// TIA Portal V17 export
// export: Created 2025-03-07T09:18:48.0864435Z, ExportSetting WithDefaults, DisplayName Totally Integrated Automation Portal, DisplayVersion V17 Update 8, DisplayName TIA Portal Openness, DisplayVersion V17 Update 8, DisplayName TIA Portal Version Control Interface, DisplayVersion V17, DisplayName SINAMICS Startdrive Advanced, DisplayVersion V17 SP2, DisplayName SINAMICS Startdrive G110M, G120, G120C, G120D, G120P, G115D, DisplayVersion V17 SP2, DisplayName SINAMICS Startdrive G130, G150, S120, S150, SINAMICS MV, S210, DisplayVersion V17 SP2, DisplayName STEP 7 Professional, DisplayVersion V17 Update 8, DisplayName SINUMERIK ONE STEP 7 Toolbox, DisplayVersion V17 Update 12, DisplayName SINUMERIK 840D sl STEP 7 Toolbox, DisplayVersion V17 Update 12, DisplayName STEP 7 Safety, DisplayVersion V17 Update 6, DisplayName WinCC Advanced, DisplayVersion V17 Update 8
FUNCTION_BLOCK "FB6500_CYLINDER"   // FB6500, LAD
{ S7_Optimized_Access := 'FALSE' }
AUTHOR : ETXETAR
VERSION : 1.0
// stored: AutoNumber false, IsIECCheckEnabled false, SetENOAutomatically false, UDAEnableTagReadback false
   VAR_INPUT
      OPTIONS_0 : Byte := 2#0000_0000;   // OPTIONS 0
      ADVANCED_1_I : Bool;   // ADVANCED 1 INPUT
      ADVANCED_2_I : Bool;   // ADVANCED 2 INPUT
      ADVANCED_3_I : Bool;   // ADVANCED 3 INPUT
      ADVANCED_4_I : Bool;   // ADVANCED 4 INPUT
      RETURNED_1_I : Bool;   // OPEN 1 INPUT
      RETURNED_2_I : Bool;   // OPEN 2 INPUT
      RETURNED_3_I : Bool;   // OPEN 3 INPUT
      RETURNED_4_I : Bool;   // OPEN 4 INPUT
      ADVANCE_CONDITIONS : Bool;   // ADVANCE CONDITIONS
      RETURN_CONDITIONS : Bool;   // OPEN CONDITIONS
      HMI_LINE_REQUEST : Bool;   // HMI LINE REQUEST
      ADVANCE_AUTO_REQUEST : Bool;   // AUTO ADVANCE REQUEST
      RETURN_AUTO_REQUEST : Bool;   // AUTO OPEN REQUEST
      UNIT_ALARM : UInt;   // UNIT NUMBER MIN. NUMBER=1 MAX. NUMBER=4
      STATION_ALARM : UInt;   // STATION NUMBER MIN. NUMBER=0 MAX. NUMBER=4
   END_VAR
   VAR_OUTPUT
      ADVANCED : Bool;   // ADVANCED
      RETURNED : Bool;   // OPEN STATUS
      ADVANCED_1_ALARM : Bool;   // ADVANCED 1 ALARM
      ADVANCED_2_ALARM : Bool;   // ADVANCED 2 ALARM
      ADVANCED_3_ALARM : Bool;   // ADVANCED 3 ALARM
      ADVANCED_4_ALARM : Bool;   // ADVANCED 4 ALARM
      RETURNED_1_ALARM : Bool;   // OPEN 1 ALARM
      RETURNED_2_ALARM : Bool;   // OPEN 2 ALARM
      RETURNED_3_ALARM : Bool;   // OPEN 3 ALARM
      RETURNED_4_ALARM : Bool;   // OPEN 4 ALARM
      HMI_MOTION_EXECUTABILITY_LEFT : Bool;   // HMI MOTION EXECUTABILITY LEFT
      HMI_MOTION_EXECUTABILITY_RIGHT : Bool;   // HMI MOTION EXECUTABILITY RIGHT
      HMI_MOTION_END_POS_LEFT : Bool;   // HMI MOTION END POSITION LEFT
      HMI_MOTION_END_POS_RIGHT : Bool;   // HMI MOTION END POSITION RIGHT
      HMI_MOTION_ACTIVE_LEFT : Bool;   // HMI MOTION ACTIVE LEFT
      HMI_MOTION_ACTIVE_RIGHT : Bool;   // HMI MOTION ACTIVE RIGHT
      ADVANCE : Bool;   // ADVANCE OUTPUT
      "RETURN" : Bool;   // OPEN OUTPUT
   END_VAR
   VAR DB_SPECIFIC
      CYL { S7_SetPoint := 'True'} : "ADVANCE_RETURN_CYL_CLADDING";
      TIMER_ADVANCED { S7_SetPoint := 'True'} : TON_TIME;   // ADVANCED TIMER
      TIMER_RETURNED { S7_SetPoint := 'True'} : TON_TIME;   // OPENED TIMER
      TIMER_SIMULTANEITY { S7_SetPoint := 'True'} : TON_TIME;   // SIMULTANEITY TIMER
      TIMER_TIME_EXCEEDED { S7_SetPoint := 'True'} : TON_TIME;   // TIME EXCEEDED TIMER
   END_VAR
   VAR_TEMP
      INPUTS_MASK : Byte;   // INPUTS_MASK
      O_BYTE_0 : Struct   // OPTIONS BYTE 0
         ADVANCED_INPUT_1 : Bool;   // ADVANCED INPUT 1 OPTION
         ADVANCED_INPUT_2 : Bool;   // ADVANCED INPUT 2 OPTION
         ADVANCED_INPUT_3 : Bool;   // ADVANCED INPUT 3 OPTION
         ADVANCED_INPUT_4 : Bool;   // ADVANCED INPUT 4 OPTION
         RETURNED_INPUT_1 : Bool;   // OPEN INPUT 1 OPTION
         RETURNED_INPUT_2 : Bool;   // OPEN INPUT 2 OPTION
         RETURNED_INPUT_3 : Bool;   // OPEN INPUT 3 OPTION
         RETURNED_INPUT_4 : Bool;   // OPEN INPUT 4 OPTION
      END_STRUCT;
      DB_NUMBER : DInt;   // DB NUMBER FOR ALARM AND HELP DECODING
   END_VAR
   // TIMER_ADVANCED.PT := T#100MS;
   // TIMER_RETURNED.PT := T#300MS;
   // TIMER_SIMULTANEITY.PT := T#100MS;
   // TIMER_TIME_EXCEEDED.PT := T#8S;
   VAR_TEMP   // added for the SCL form of the ladder/FBD networks
      _w1 : Bool;
      _w2 : Bool;
   END_VAR
BEGIN

NETWORK
TITLE = READ INSTANCE DB
      L     DINO;
      +     10#800000;
      T     #DB_NUMBER;


REGION Network 2: OPTIONS
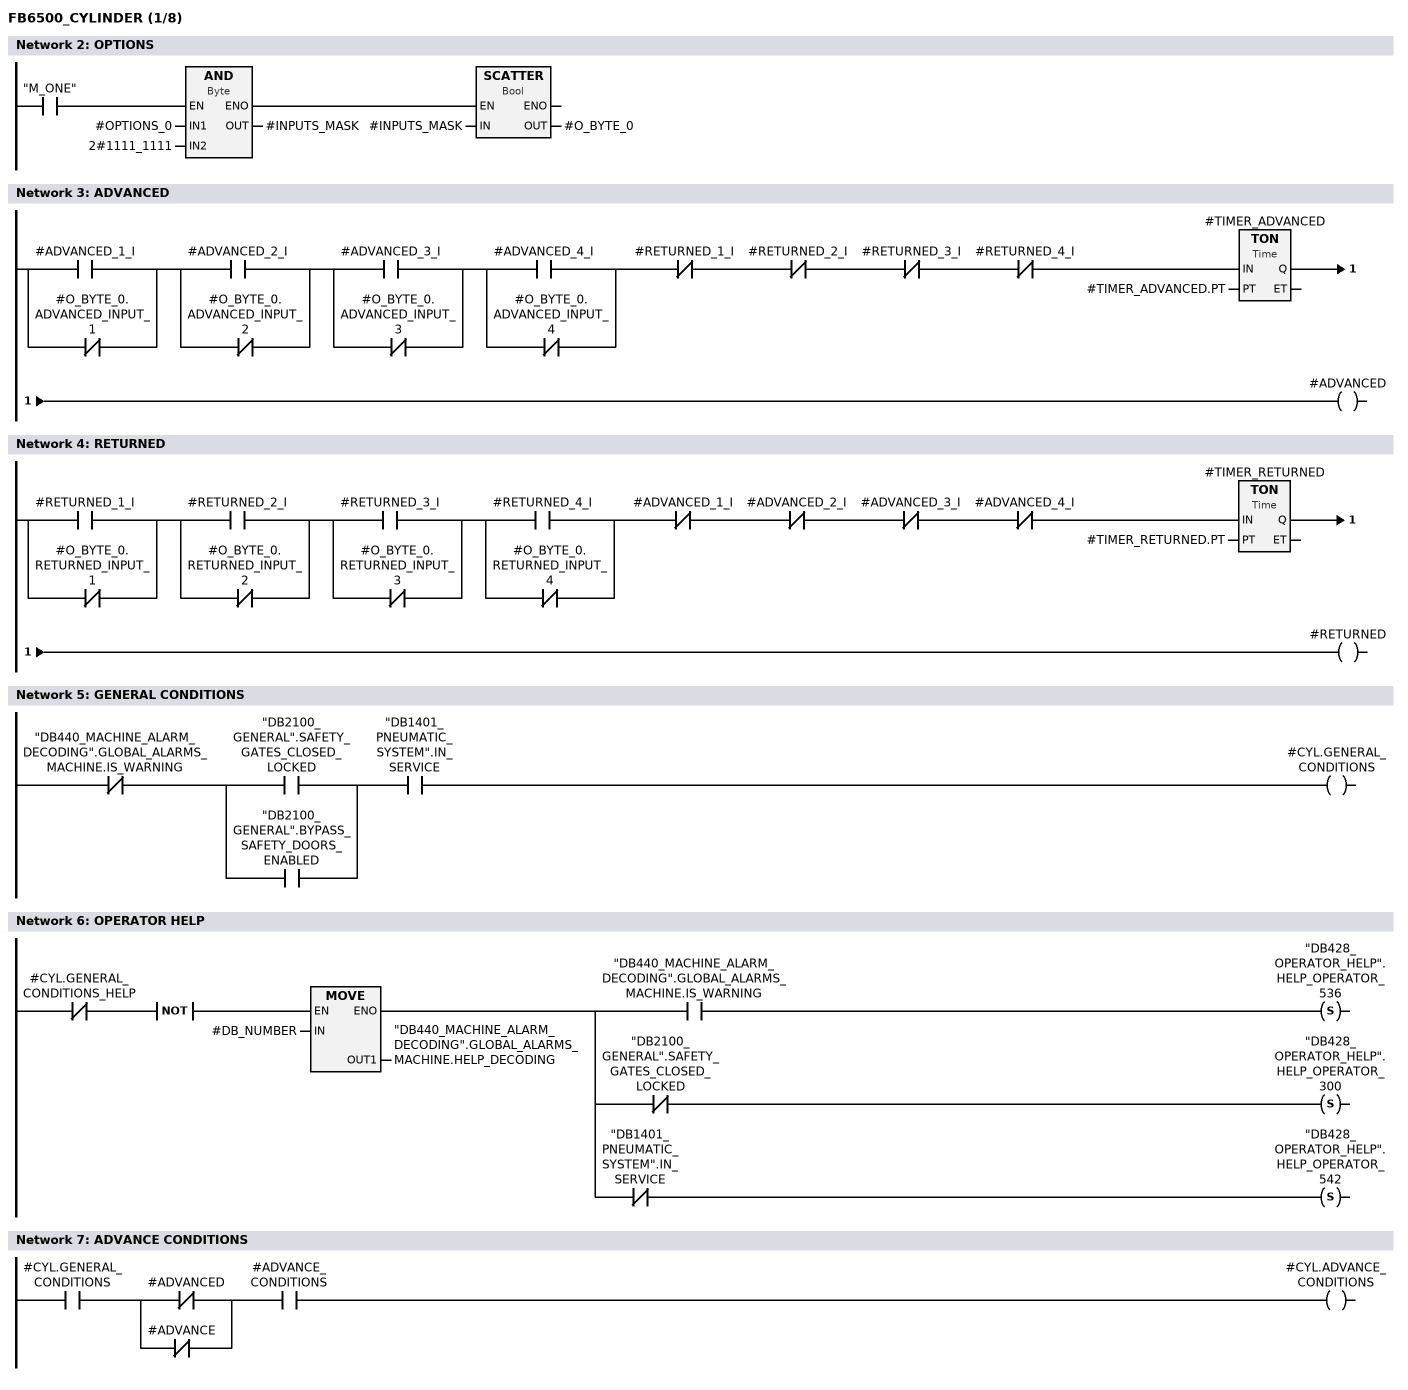
   RUNG wire#powerrail
      Contact( "M_ONE" )
      { S7_Templates := "SrcType := Byte"; S7_GenerateENO := "TRUE" } And(in1 := #OPTIONS_0, in2 := 2#1111_1111, out => #INPUTS_MASK)
      { S7_Templates := "[dest_type := Bool, src_type := Byte]" } SCATTER(IN := #INPUTS_MASK, OUT => #O_BYTE_0)
   END_RUNG
   // the same network as SCL:
   IF "M_ONE" THEN
       #INPUTS_MASK := #OPTIONS_0 AND 2#1111_1111;
       SCATTER(IN := #INPUTS_MASK, OUT => #O_BYTE_0);
   END_IF;
END_REGION

REGION Network 3: ADVANCED
   RUNG wire#powerrail
      Contact( #ADVANCED_1_I )
      wire#w1
      Contact( #ADVANCED_2_I )
      wire#w2
      Contact( #ADVANCED_3_I )
      wire#w3
      Contact( #ADVANCED_4_I )
      wire#w4
      I_Contact( #RETURNED_1_I )
      I_Contact( #RETURNED_2_I )
      I_Contact( #RETURNED_3_I )
      I_Contact( #RETURNED_4_I )
      { S7_Templates := "time_type := Time" } #TIMER_ADVANCED.TON(pt := #TIMER_ADVANCED.PT, et =>)
      Coil( #ADVANCED )
   END_RUNG
   RUNG wire#powerrail
      I_Contact( #O_BYTE_0.ADVANCED_INPUT_1 )
   END_RUNG wire#w1
   RUNG wire#w1
      I_Contact( #O_BYTE_0.ADVANCED_INPUT_2 )
   END_RUNG wire#w2
   RUNG wire#w2
      I_Contact( #O_BYTE_0.ADVANCED_INPUT_3 )
   END_RUNG wire#w3
   RUNG wire#w3
      I_Contact( #O_BYTE_0.ADVANCED_INPUT_4 )
   END_RUNG wire#w4
   // the same network as SCL:
   #TIMER_ADVANCED(IN := (#ADVANCED_1_I OR NOT #O_BYTE_0.ADVANCED_INPUT_1) AND (#ADVANCED_2_I OR NOT #O_BYTE_0.ADVANCED_INPUT_2) AND (#ADVANCED_3_I OR NOT #O_BYTE_0.ADVANCED_INPUT_3) AND (#ADVANCED_4_I OR NOT #O_BYTE_0.ADVANCED_INPUT_4) AND NOT #RETURNED_1_I AND NOT #RETURNED_2_I AND NOT #RETURNED_3_I AND NOT #RETURNED_4_I,   // TON
                   PT := #TIMER_ADVANCED.PT);
   #ADVANCED := #TIMER_ADVANCED.Q;
END_REGION

REGION Network 4: RETURNED
   RUNG wire#powerrail
      Contact( #RETURNED_1_I )
      wire#w1
      Contact( #RETURNED_2_I )
      wire#w2
      Contact( #RETURNED_3_I )
      wire#w3
      Contact( #RETURNED_4_I )
      wire#w4
      I_Contact( #ADVANCED_1_I )
      I_Contact( #ADVANCED_2_I )
      I_Contact( #ADVANCED_3_I )
      I_Contact( #ADVANCED_4_I )
      { S7_Templates := "time_type := Time" } #TIMER_RETURNED.TON(pt := #TIMER_RETURNED.PT, et =>)
      Coil( #RETURNED )
   END_RUNG
   RUNG wire#powerrail
      I_Contact( #O_BYTE_0.RETURNED_INPUT_1 )
   END_RUNG wire#w1
   RUNG wire#w1
      I_Contact( #O_BYTE_0.RETURNED_INPUT_2 )
   END_RUNG wire#w2
   RUNG wire#w2
      I_Contact( #O_BYTE_0.RETURNED_INPUT_3 )
   END_RUNG wire#w3
   RUNG wire#w3
      I_Contact( #O_BYTE_0.RETURNED_INPUT_4 )
   END_RUNG wire#w4
   // the same network as SCL:
   #TIMER_RETURNED(IN := (#RETURNED_1_I OR NOT #O_BYTE_0.RETURNED_INPUT_1) AND (#RETURNED_2_I OR NOT #O_BYTE_0.RETURNED_INPUT_2) AND (#RETURNED_3_I OR NOT #O_BYTE_0.RETURNED_INPUT_3) AND (#RETURNED_4_I OR NOT #O_BYTE_0.RETURNED_INPUT_4) AND NOT #ADVANCED_1_I AND NOT #ADVANCED_2_I AND NOT #ADVANCED_3_I AND NOT #ADVANCED_4_I,   // TON
                   PT := #TIMER_RETURNED.PT);
   #RETURNED := #TIMER_RETURNED.Q;
END_REGION

REGION Network 5: GENERAL CONDITIONS
   RUNG wire#powerrail
      I_Contact( "DB440_MACHINE_ALARM_DECODING".GLOBAL_ALARMS_MACHINE.IS_WARNING )
      wire#w1
      Contact( "DB2100_GENERAL".SAFETY_GATES_CLOSED_LOCKED )
      wire#w2
      Contact( "DB1401_PNEUMATIC_SYSTEM".IN_SERVICE )
      Coil( #CYL.GENERAL_CONDITIONS )
   END_RUNG
   RUNG wire#w1
      Contact( "DB2100_GENERAL".BYPASS_SAFETY_DOORS_ENABLED )
   END_RUNG wire#w2
   // the same network as SCL:
   #CYL.GENERAL_CONDITIONS := NOT "DB440_MACHINE_ALARM_DECODING".GLOBAL_ALARMS_MACHINE.IS_WARNING AND ("DB2100_GENERAL".SAFETY_GATES_CLOSED_LOCKED OR "DB2100_GENERAL".BYPASS_SAFETY_DOORS_ENABLED) AND "DB1401_PNEUMATIC_SYSTEM".IN_SERVICE;
END_REGION

REGION Network 6: OPERATOR HELP
   RUNG wire#powerrail
      I_Contact( #CYL.GENERAL_CONDITIONS_HELP )
      Not()
      { S7_GenerateENO := "TRUE" } Move(in := #DB_NUMBER, out1 => "DB440_MACHINE_ALARM_DECODING".GLOBAL_ALARMS_MACHINE.HELP_DECODING)
      wire#w1
      Contact( "DB440_MACHINE_ALARM_DECODING".GLOBAL_ALARMS_MACHINE.IS_WARNING )
      S_Coil( "DB428_OPERATOR_HELP".HELP_OPERATOR_536 )
   END_RUNG
   RUNG wire#w1
      I_Contact( "DB2100_GENERAL".SAFETY_GATES_CLOSED_LOCKED )
      S_Coil( "DB428_OPERATOR_HELP".HELP_OPERATOR_300 )
   END_RUNG
   RUNG wire#w1
      I_Contact( "DB1401_PNEUMATIC_SYSTEM".IN_SERVICE )
      S_Coil( "DB428_OPERATOR_HELP".HELP_OPERATOR_542 )
   END_RUNG
   // the same network as SCL:
   // ENO of a box is taken as its EN; it also drops when the box reports an error
   #_w1 := NOT (NOT #CYL.GENERAL_CONDITIONS_HELP);
   IF #_w1 THEN "DB440_MACHINE_ALARM_DECODING".GLOBAL_ALARMS_MACHINE.HELP_DECODING := #DB_NUMBER; END_IF;
   IF #_w1 AND "DB440_MACHINE_ALARM_DECODING".GLOBAL_ALARMS_MACHINE.IS_WARNING THEN
       "DB428_OPERATOR_HELP".HELP_OPERATOR_536 := TRUE;
   END_IF;
   IF #_w1 AND NOT "DB2100_GENERAL".SAFETY_GATES_CLOSED_LOCKED THEN
       "DB428_OPERATOR_HELP".HELP_OPERATOR_300 := TRUE;
   END_IF;
   IF #_w1 AND NOT "DB1401_PNEUMATIC_SYSTEM".IN_SERVICE THEN
       "DB428_OPERATOR_HELP".HELP_OPERATOR_542 := TRUE;
   END_IF;
END_REGION

REGION Network 7: ADVANCE CONDITIONS
   RUNG wire#powerrail
      Contact( #CYL.GENERAL_CONDITIONS )
      wire#w1
      I_Contact( #ADVANCED )
      wire#w2
      Contact( #ADVANCE_CONDITIONS )
      Coil( #CYL.ADVANCE_CONDITIONS )
   END_RUNG
   RUNG wire#w1
      I_Contact( #ADVANCE )
   END_RUNG wire#w2
   // the same network as SCL:
   #CYL.ADVANCE_CONDITIONS := #CYL.GENERAL_CONDITIONS AND (NOT #ADVANCED OR NOT #ADVANCE) AND #ADVANCE_CONDITIONS;
END_REGION

REGION Network 8: OPERATOR HELP
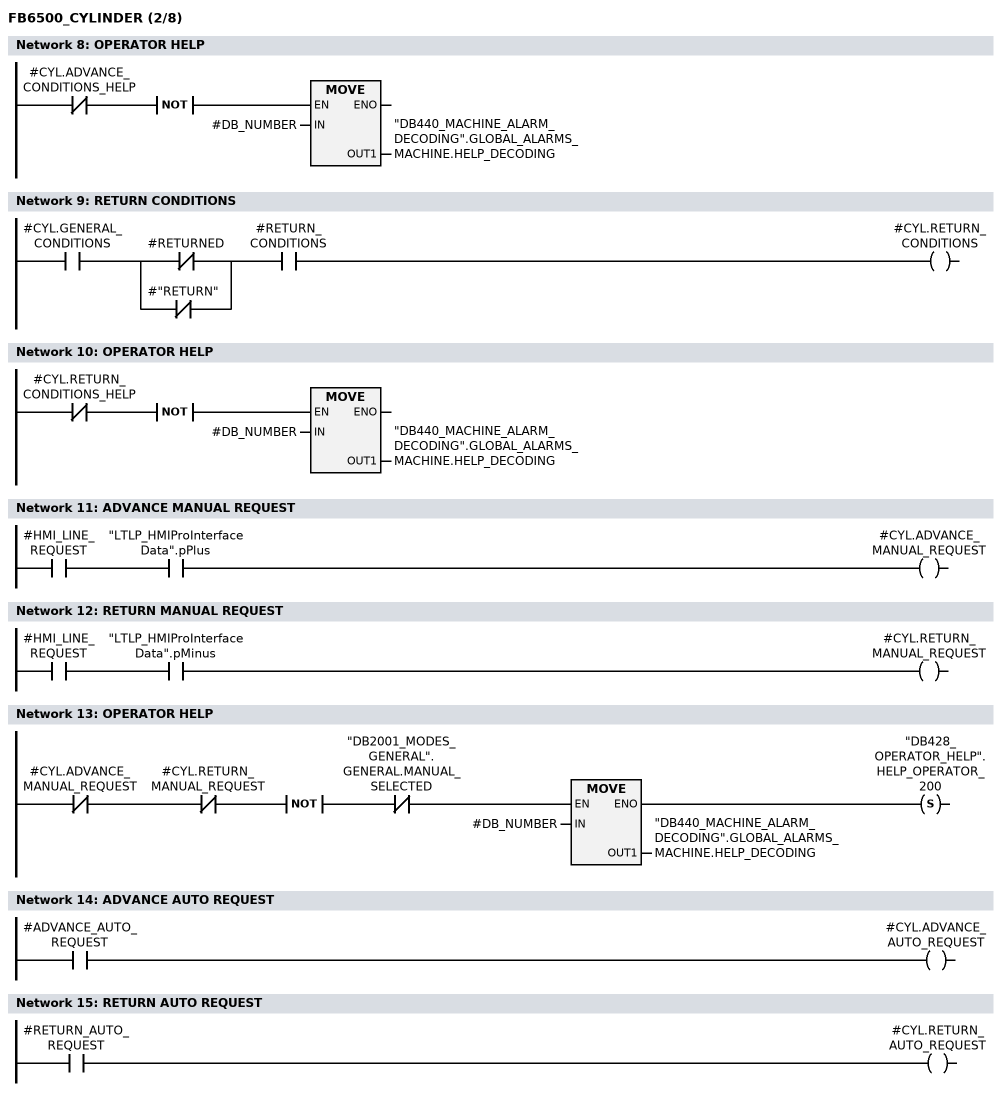
   RUNG wire#powerrail
      I_Contact( #CYL.ADVANCE_CONDITIONS_HELP )
      Not()
      { S7_GenerateENO := "TRUE" } Move(in := #DB_NUMBER, out1 => "DB440_MACHINE_ALARM_DECODING".GLOBAL_ALARMS_MACHINE.HELP_DECODING)
   END_RUNG
   // the same network as SCL:
   IF NOT (NOT #CYL.ADVANCE_CONDITIONS_HELP) THEN
       "DB440_MACHINE_ALARM_DECODING".GLOBAL_ALARMS_MACHINE.HELP_DECODING := #DB_NUMBER;
   END_IF;
END_REGION

REGION Network 9: RETURN CONDITIONS
   RUNG wire#powerrail
      Contact( #CYL.GENERAL_CONDITIONS )
      wire#w1
      I_Contact( #RETURNED )
      wire#w2
      Contact( #RETURN_CONDITIONS )
      Coil( #CYL.RETURN_CONDITIONS )
   END_RUNG
   RUNG wire#w1
      I_Contact( #"RETURN" )
   END_RUNG wire#w2
   // the same network as SCL:
   #CYL.RETURN_CONDITIONS := #CYL.GENERAL_CONDITIONS AND (NOT #RETURNED OR NOT #"RETURN") AND #RETURN_CONDITIONS;
END_REGION

REGION Network 10: OPERATOR HELP
   RUNG wire#powerrail
      I_Contact( #CYL.RETURN_CONDITIONS_HELP )
      Not()
      { S7_GenerateENO := "TRUE" } Move(in := #DB_NUMBER, out1 => "DB440_MACHINE_ALARM_DECODING".GLOBAL_ALARMS_MACHINE.HELP_DECODING)
   END_RUNG
   // the same network as SCL:
   IF NOT (NOT #CYL.RETURN_CONDITIONS_HELP) THEN
       "DB440_MACHINE_ALARM_DECODING".GLOBAL_ALARMS_MACHINE.HELP_DECODING := #DB_NUMBER;
   END_IF;
END_REGION

REGION Network 11: ADVANCE MANUAL REQUEST
   RUNG wire#powerrail
      Contact( #HMI_LINE_REQUEST )
      Contact( "LTLP_HMIProInterfaceData".pPlus )
      Coil( #CYL.ADVANCE_MANUAL_REQUEST )
   END_RUNG
   // the same network as SCL:
   #CYL.ADVANCE_MANUAL_REQUEST := #HMI_LINE_REQUEST AND "LTLP_HMIProInterfaceData".pPlus;
END_REGION

REGION Network 12: RETURN MANUAL REQUEST
   RUNG wire#powerrail
      Contact( #HMI_LINE_REQUEST )
      Contact( "LTLP_HMIProInterfaceData".pMinus )
      Coil( #CYL.RETURN_MANUAL_REQUEST )
   END_RUNG
   // the same network as SCL:
   #CYL.RETURN_MANUAL_REQUEST := #HMI_LINE_REQUEST AND "LTLP_HMIProInterfaceData".pMinus;
END_REGION

REGION Network 13: OPERATOR HELP
   RUNG wire#powerrail
      I_Contact( #CYL.ADVANCE_MANUAL_REQUEST )
      I_Contact( #CYL.RETURN_MANUAL_REQUEST )
      Not()
      I_Contact( "DB2001_MODES_GENERAL".GENERAL.MANUAL_SELECTED )
      { S7_GenerateENO := "TRUE" } Move(in := #DB_NUMBER, out1 => "DB440_MACHINE_ALARM_DECODING".GLOBAL_ALARMS_MACHINE.HELP_DECODING)
      S_Coil( "DB428_OPERATOR_HELP".HELP_OPERATOR_200 )
   END_RUNG
   // the same network as SCL:
   // ENO of a box is taken as its EN; it also drops when the box reports an error
   IF NOT (NOT #CYL.ADVANCE_MANUAL_REQUEST AND NOT #CYL.RETURN_MANUAL_REQUEST) AND NOT "DB2001_MODES_GENERAL".GENERAL.MANUAL_SELECTED THEN
       "DB440_MACHINE_ALARM_DECODING".GLOBAL_ALARMS_MACHINE.HELP_DECODING := #DB_NUMBER;
       "DB428_OPERATOR_HELP".HELP_OPERATOR_200 := TRUE;
   END_IF;
END_REGION

REGION Network 14: ADVANCE AUTO REQUEST
   RUNG wire#powerrail
      Contact( #ADVANCE_AUTO_REQUEST )
      Coil( #CYL.ADVANCE_AUTO_REQUEST )
   END_RUNG
   // the same network as SCL:
   #CYL.ADVANCE_AUTO_REQUEST := #ADVANCE_AUTO_REQUEST;
END_REGION

REGION Network 15: RETURN AUTO REQUEST
   RUNG wire#powerrail
      Contact( #RETURN_AUTO_REQUEST )
      Coil( #CYL.RETURN_AUTO_REQUEST )
   END_RUNG
   // the same network as SCL:
   #CYL.RETURN_AUTO_REQUEST := #RETURN_AUTO_REQUEST;
END_REGION

REGION Network 16: ADVANCE GLOBAL REQUEST
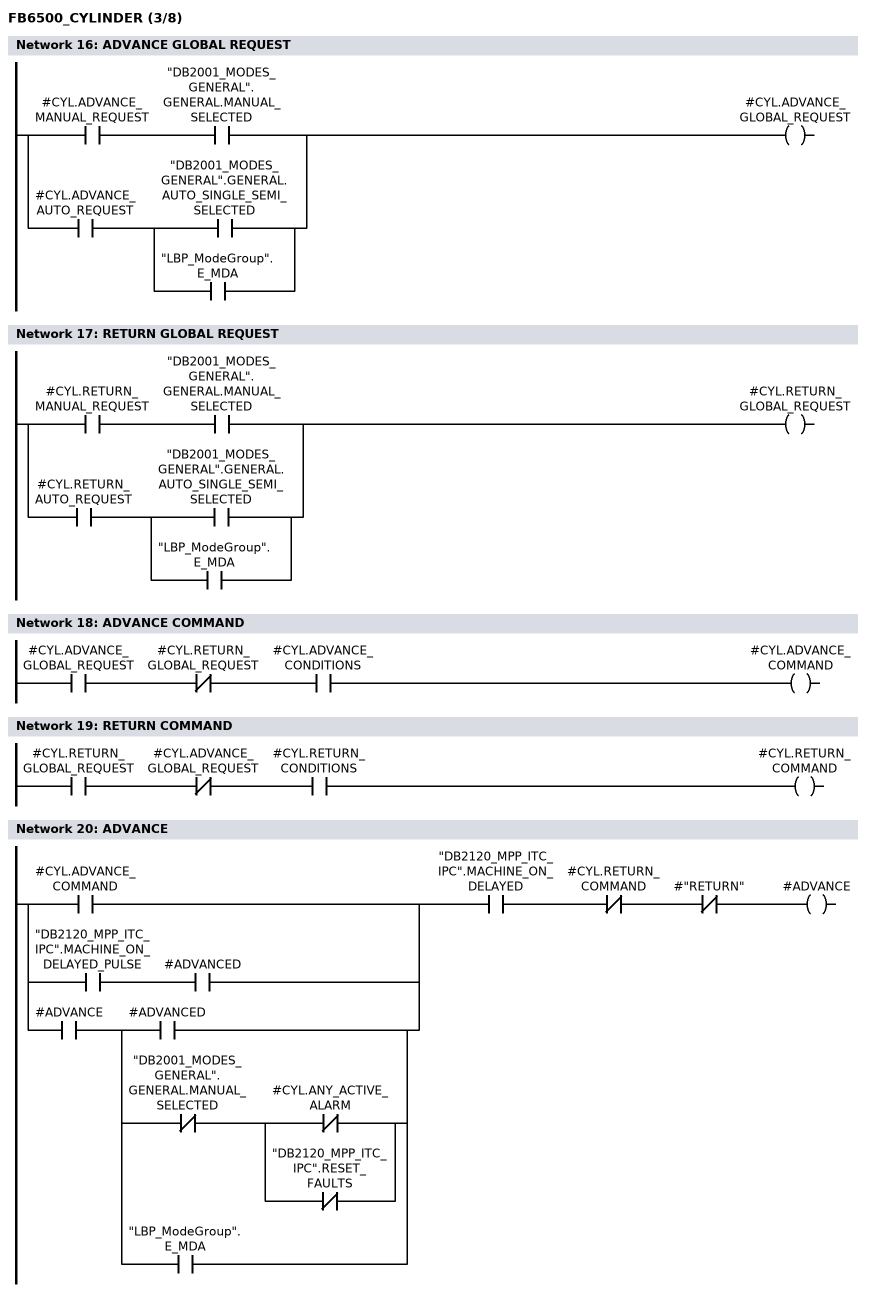
   RUNG wire#powerrail
      Contact( #CYL.ADVANCE_MANUAL_REQUEST )
      Contact( "DB2001_MODES_GENERAL".GENERAL.MANUAL_SELECTED )
      wire#w1
      Coil( #CYL.ADVANCE_GLOBAL_REQUEST )
   END_RUNG
   RUNG wire#powerrail
      Contact( #CYL.ADVANCE_AUTO_REQUEST )
      wire#w2
      Contact( "DB2001_MODES_GENERAL".GENERAL.AUTO_SINGLE_SEMI_SELECTED )
   END_RUNG wire#w1
   RUNG wire#w2
      Contact( "LBP_ModeGroup".E_MDA )
   END_RUNG wire#w1
   // the same network as SCL:
   #CYL.ADVANCE_GLOBAL_REQUEST := (#CYL.ADVANCE_MANUAL_REQUEST AND "DB2001_MODES_GENERAL".GENERAL.MANUAL_SELECTED) OR (#CYL.ADVANCE_AUTO_REQUEST AND ("DB2001_MODES_GENERAL".GENERAL.AUTO_SINGLE_SEMI_SELECTED OR "LBP_ModeGroup".E_MDA));
END_REGION

REGION Network 17: RETURN GLOBAL REQUEST
   RUNG wire#powerrail
      Contact( #CYL.RETURN_MANUAL_REQUEST )
      Contact( "DB2001_MODES_GENERAL".GENERAL.MANUAL_SELECTED )
      wire#w1
      Coil( #CYL.RETURN_GLOBAL_REQUEST )
   END_RUNG
   RUNG wire#powerrail
      Contact( #CYL.RETURN_AUTO_REQUEST )
      wire#w2
      Contact( "DB2001_MODES_GENERAL".GENERAL.AUTO_SINGLE_SEMI_SELECTED )
   END_RUNG wire#w1
   RUNG wire#w2
      Contact( "LBP_ModeGroup".E_MDA )
   END_RUNG wire#w1
   // the same network as SCL:
   #CYL.RETURN_GLOBAL_REQUEST := (#CYL.RETURN_MANUAL_REQUEST AND "DB2001_MODES_GENERAL".GENERAL.MANUAL_SELECTED) OR (#CYL.RETURN_AUTO_REQUEST AND ("DB2001_MODES_GENERAL".GENERAL.AUTO_SINGLE_SEMI_SELECTED OR "LBP_ModeGroup".E_MDA));
END_REGION

REGION Network 18: ADVANCE COMMAND
   RUNG wire#powerrail
      Contact( #CYL.ADVANCE_GLOBAL_REQUEST )
      I_Contact( #CYL.RETURN_GLOBAL_REQUEST )
      Contact( #CYL.ADVANCE_CONDITIONS )
      Coil( #CYL.ADVANCE_COMMAND )
   END_RUNG
   // the same network as SCL:
   #CYL.ADVANCE_COMMAND := #CYL.ADVANCE_GLOBAL_REQUEST AND NOT #CYL.RETURN_GLOBAL_REQUEST AND #CYL.ADVANCE_CONDITIONS;
END_REGION

REGION Network 19: RETURN COMMAND
   RUNG wire#powerrail
      Contact( #CYL.RETURN_GLOBAL_REQUEST )
      I_Contact( #CYL.ADVANCE_GLOBAL_REQUEST )
      Contact( #CYL.RETURN_CONDITIONS )
      Coil( #CYL.RETURN_COMMAND )
   END_RUNG
   // the same network as SCL:
   #CYL.RETURN_COMMAND := #CYL.RETURN_GLOBAL_REQUEST AND NOT #CYL.ADVANCE_GLOBAL_REQUEST AND #CYL.RETURN_CONDITIONS;
END_REGION

REGION Network 20: ADVANCE
   RUNG wire#powerrail
      Contact( #CYL.ADVANCE_COMMAND )
      wire#w1
      Contact( "DB2120_MPP_ITC_IPC".MACHINE_ON_DELAYED )
      I_Contact( #CYL.RETURN_COMMAND )
      I_Contact( #"RETURN" )
      Coil( #ADVANCE )
   END_RUNG
   RUNG wire#powerrail
      Contact( "DB2120_MPP_ITC_IPC".MACHINE_ON_DELAYED_PULSE )
      Contact( #ADVANCED )
   END_RUNG wire#w1
   RUNG wire#powerrail
      Contact( #ADVANCE )
      wire#w2
      Contact( #ADVANCED )
   END_RUNG wire#w1
   RUNG wire#w2
      I_Contact( "DB2001_MODES_GENERAL".GENERAL.MANUAL_SELECTED )
      wire#w3
      I_Contact( #CYL.ANY_ACTIVE_ALARM )
   END_RUNG wire#w1
   RUNG wire#w3
      I_Contact( "DB2120_MPP_ITC_IPC".RESET_FAULTS )
   END_RUNG wire#w1
   RUNG wire#w2
      Contact( "LBP_ModeGroup".E_MDA )
   END_RUNG wire#w1
   // the same network as SCL:
   #ADVANCE := (#CYL.ADVANCE_COMMAND OR ("DB2120_MPP_ITC_IPC".MACHINE_ON_DELAYED_PULSE AND #ADVANCED) OR (#ADVANCE AND (#ADVANCED OR (NOT "DB2001_MODES_GENERAL".GENERAL.MANUAL_SELECTED AND (NOT #CYL.ANY_ACTIVE_ALARM OR NOT "DB2120_MPP_ITC_IPC".RESET_FAULTS)) OR "LBP_ModeGroup".E_MDA))) AND "DB2120_MPP_ITC_IPC".MACHINE_ON_DELAYED AND NOT #CYL.RETURN_COMMAND AND NOT #"RETURN";
END_REGION

REGION Network 21: RETURN
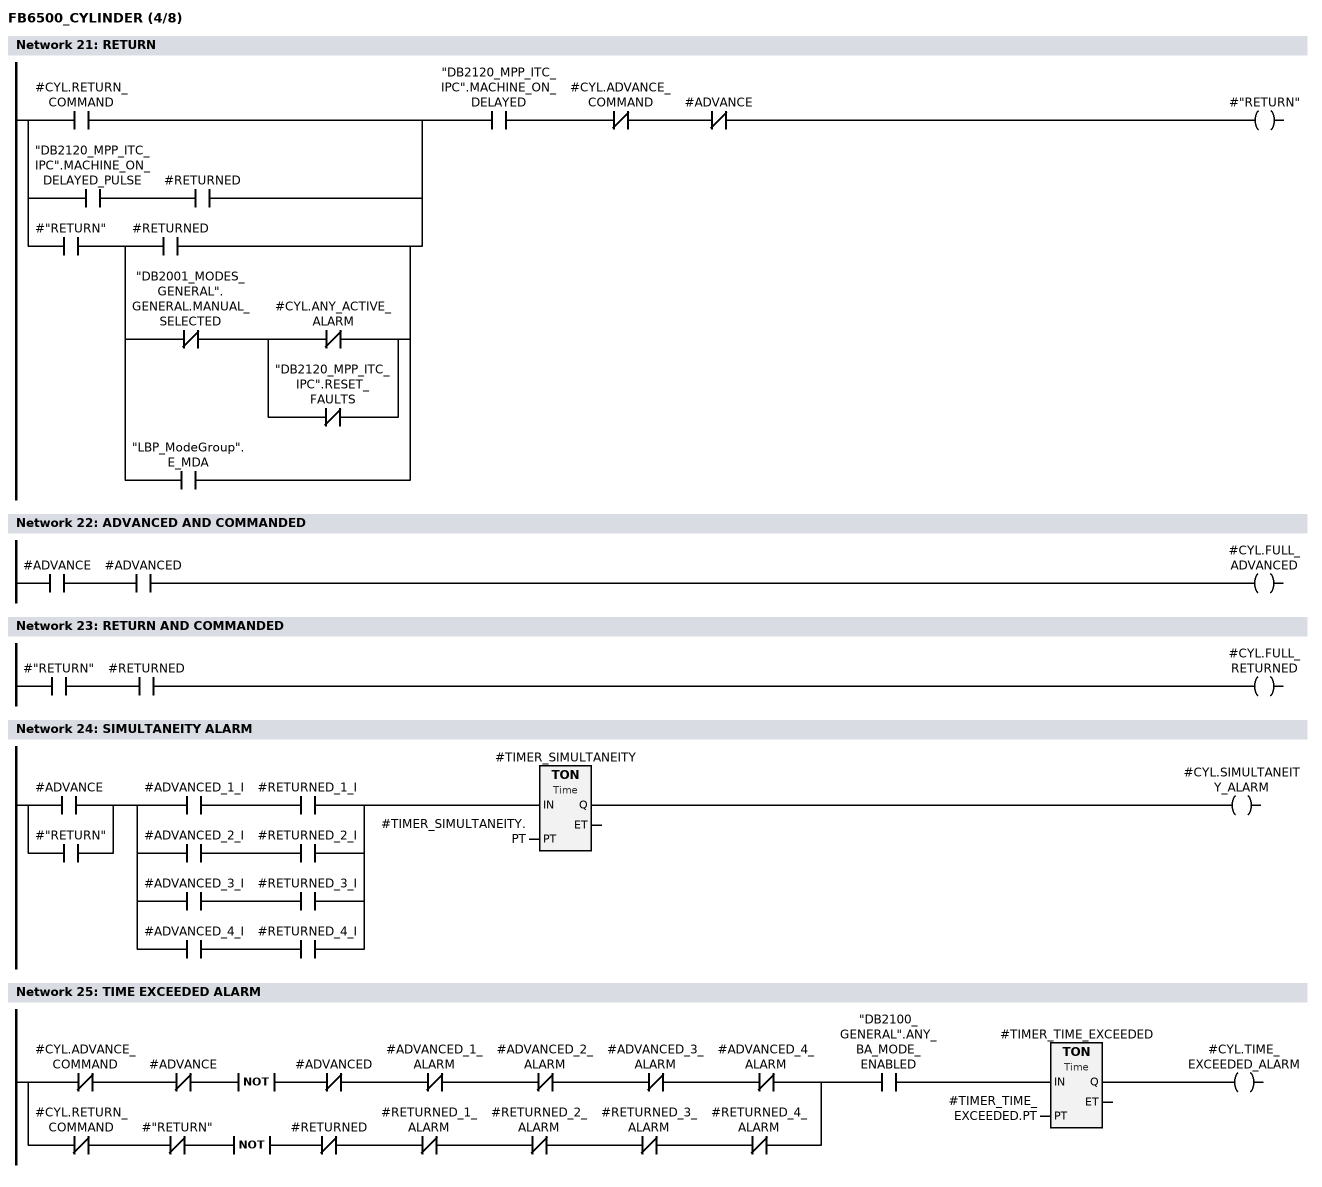
   RUNG wire#powerrail
      Contact( #CYL.RETURN_COMMAND )
      wire#w1
      Contact( "DB2120_MPP_ITC_IPC".MACHINE_ON_DELAYED )
      I_Contact( #CYL.ADVANCE_COMMAND )
      I_Contact( #ADVANCE )
      Coil( #"RETURN" )
   END_RUNG
   RUNG wire#powerrail
      Contact( "DB2120_MPP_ITC_IPC".MACHINE_ON_DELAYED_PULSE )
      Contact( #RETURNED )
   END_RUNG wire#w1
   RUNG wire#powerrail
      Contact( #"RETURN" )
      wire#w2
      Contact( #RETURNED )
   END_RUNG wire#w1
   RUNG wire#w2
      I_Contact( "DB2001_MODES_GENERAL".GENERAL.MANUAL_SELECTED )
      wire#w3
      I_Contact( #CYL.ANY_ACTIVE_ALARM )
   END_RUNG wire#w1
   RUNG wire#w3
      I_Contact( "DB2120_MPP_ITC_IPC".RESET_FAULTS )
   END_RUNG wire#w1
   RUNG wire#w2
      Contact( "LBP_ModeGroup".E_MDA )
   END_RUNG wire#w1
   // the same network as SCL:
   #"RETURN" := (#CYL.RETURN_COMMAND OR ("DB2120_MPP_ITC_IPC".MACHINE_ON_DELAYED_PULSE AND #RETURNED) OR (#"RETURN" AND (#RETURNED OR (NOT "DB2001_MODES_GENERAL".GENERAL.MANUAL_SELECTED AND (NOT #CYL.ANY_ACTIVE_ALARM OR NOT "DB2120_MPP_ITC_IPC".RESET_FAULTS)) OR "LBP_ModeGroup".E_MDA))) AND "DB2120_MPP_ITC_IPC".MACHINE_ON_DELAYED AND NOT #CYL.ADVANCE_COMMAND AND NOT #ADVANCE;
END_REGION

REGION Network 22: ADVANCED AND COMMANDED
   RUNG wire#powerrail
      Contact( #ADVANCE )
      Contact( #ADVANCED )
      Coil( #CYL.FULL_ADVANCED )
   END_RUNG
   // the same network as SCL:
   #CYL.FULL_ADVANCED := #ADVANCE AND #ADVANCED;
END_REGION

REGION Network 23: RETURN AND COMMANDED
   RUNG wire#powerrail
      Contact( #"RETURN" )
      Contact( #RETURNED )
      Coil( #CYL.FULL_RETURNED )
   END_RUNG
   // the same network as SCL:
   #CYL.FULL_RETURNED := #"RETURN" AND #RETURNED;
END_REGION

REGION Network 24: SIMULTANEITY ALARM
   RUNG wire#powerrail
      Contact( #ADVANCE )
      wire#w1
      Contact( #ADVANCED_1_I )
      Contact( #RETURNED_1_I )
      wire#w2
      { S7_Templates := "time_type := Time" } #TIMER_SIMULTANEITY.TON(pt := #TIMER_SIMULTANEITY.PT, et =>)
      Coil( #CYL.SIMULTANEITY_ALARM )
   END_RUNG
   RUNG wire#powerrail
      Contact( #"RETURN" )
   END_RUNG wire#w1
   RUNG wire#w1
      Contact( #ADVANCED_2_I )
      Contact( #RETURNED_2_I )
   END_RUNG wire#w2
   RUNG wire#w1
      Contact( #ADVANCED_3_I )
      Contact( #RETURNED_3_I )
   END_RUNG wire#w2
   RUNG wire#w1
      Contact( #ADVANCED_4_I )
      Contact( #RETURNED_4_I )
   END_RUNG wire#w2
   // the same network as SCL:
   #TIMER_SIMULTANEITY(IN := (#ADVANCE OR #"RETURN") AND ((#ADVANCED_1_I AND #RETURNED_1_I) OR (#ADVANCED_2_I AND #RETURNED_2_I) OR (#ADVANCED_3_I AND #RETURNED_3_I) OR (#ADVANCED_4_I AND #RETURNED_4_I)),   // TON
                       PT := #TIMER_SIMULTANEITY.PT);
   #CYL.SIMULTANEITY_ALARM := #TIMER_SIMULTANEITY.Q;
END_REGION

REGION Network 25: TIME EXCEEDED ALARM
   RUNG wire#powerrail
      I_Contact( #CYL.ADVANCE_COMMAND )
      I_Contact( #ADVANCE )
      Not()
      I_Contact( #ADVANCED )
      I_Contact( #ADVANCED_1_ALARM )
      I_Contact( #ADVANCED_2_ALARM )
      I_Contact( #ADVANCED_3_ALARM )
      I_Contact( #ADVANCED_4_ALARM )
      wire#w1
      Contact( "DB2100_GENERAL".ANY_BA_MODE_ENABLED )
      { S7_Templates := "time_type := Time" } #TIMER_TIME_EXCEEDED.TON(pt := #TIMER_TIME_EXCEEDED.PT, et =>)
      Coil( #CYL.TIME_EXCEEDED_ALARM )
   END_RUNG
   RUNG wire#powerrail
      I_Contact( #CYL.RETURN_COMMAND )
      I_Contact( #"RETURN" )
      Not()
      I_Contact( #RETURNED )
      I_Contact( #RETURNED_1_ALARM )
      I_Contact( #RETURNED_2_ALARM )
      I_Contact( #RETURNED_3_ALARM )
      I_Contact( #RETURNED_4_ALARM )
   END_RUNG wire#w1
   // the same network as SCL:
   #TIMER_TIME_EXCEEDED(IN := ((NOT (NOT #CYL.ADVANCE_COMMAND AND NOT #ADVANCE) AND NOT #ADVANCED AND NOT #ADVANCED_1_ALARM AND NOT #ADVANCED_2_ALARM AND NOT #ADVANCED_3_ALARM AND NOT #ADVANCED_4_ALARM) OR (NOT (NOT #CYL.RETURN_COMMAND AND NOT #"RETURN") AND NOT #RETURNED AND NOT #RETURNED_1_ALARM AND NOT #RETURNED_2_ALARM AND NOT #RETURNED_3_ALARM AND NOT #RETURNED_4_ALARM)) AND "DB2100_GENERAL".ANY_BA_MODE_ENABLED,   // TON
                        PT := #TIMER_TIME_EXCEEDED.PT);
   #CYL.TIME_EXCEEDED_ALARM := #TIMER_TIME_EXCEEDED.Q;
END_REGION

REGION Network 26: ADVANCED 1 ALARM
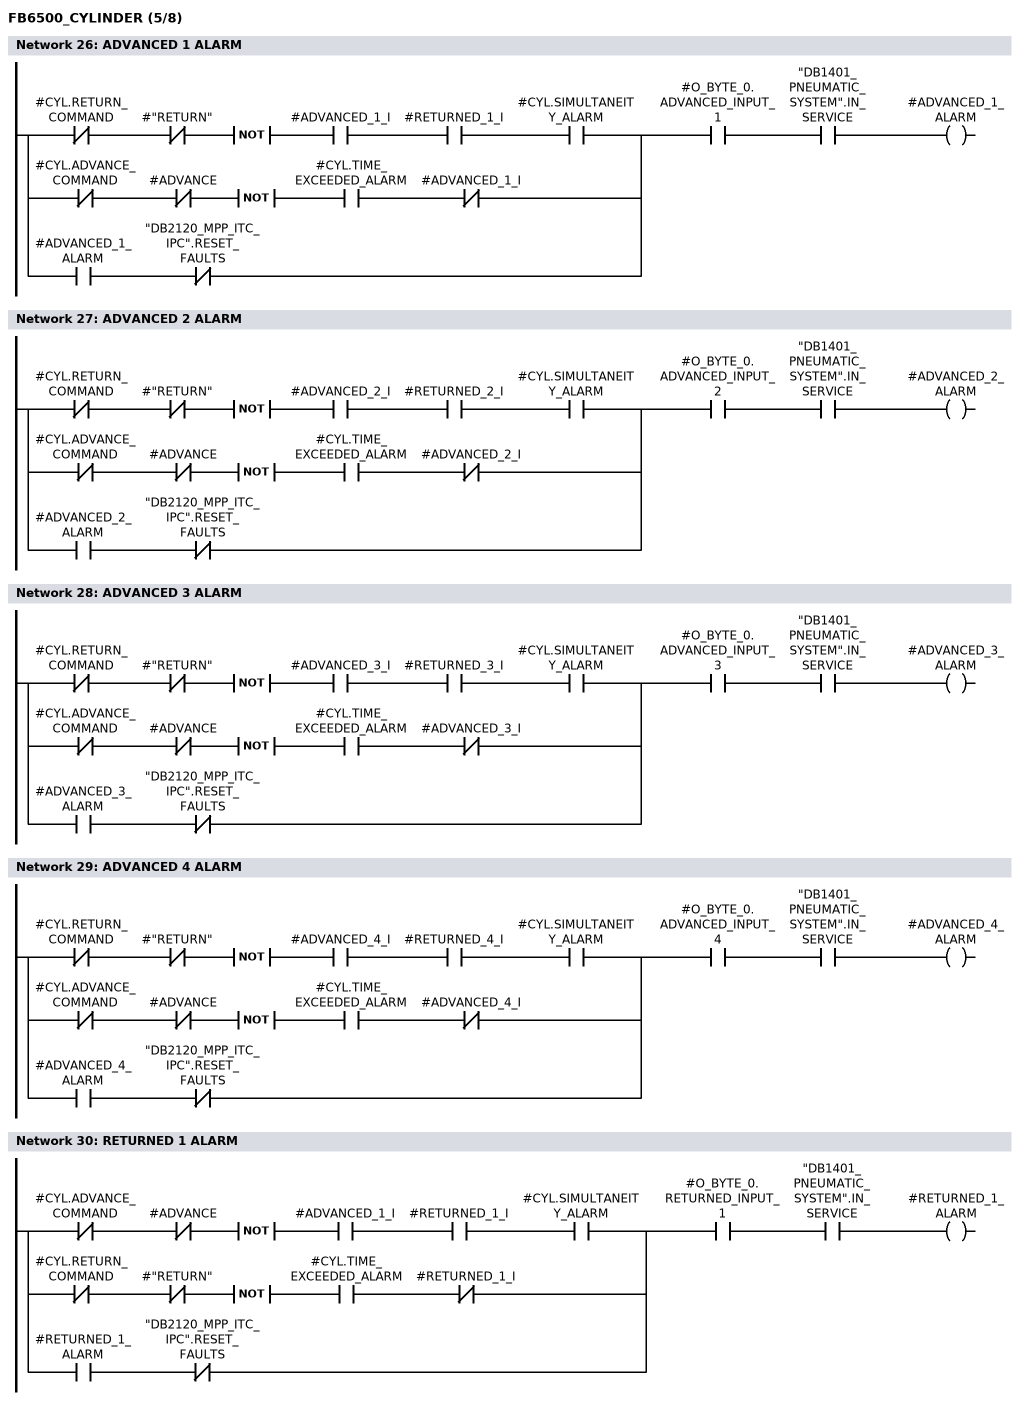
   RUNG wire#powerrail
      I_Contact( #CYL.RETURN_COMMAND )
      I_Contact( #"RETURN" )
      Not()
      Contact( #ADVANCED_1_I )
      Contact( #RETURNED_1_I )
      Contact( #CYL.SIMULTANEITY_ALARM )
      wire#w1
      Contact( #O_BYTE_0.ADVANCED_INPUT_1 )
      Contact( "DB1401_PNEUMATIC_SYSTEM".IN_SERVICE )
      Coil( #ADVANCED_1_ALARM )
   END_RUNG
   RUNG wire#powerrail
      I_Contact( #CYL.ADVANCE_COMMAND )
      I_Contact( #ADVANCE )
      Not()
      Contact( #CYL.TIME_EXCEEDED_ALARM )
      I_Contact( #ADVANCED_1_I )
   END_RUNG wire#w1
   RUNG wire#powerrail
      Contact( #ADVANCED_1_ALARM )
      I_Contact( "DB2120_MPP_ITC_IPC".RESET_FAULTS )
   END_RUNG wire#w1
   // the same network as SCL:
   #ADVANCED_1_ALARM := ((NOT (NOT #CYL.RETURN_COMMAND AND NOT #"RETURN") AND #ADVANCED_1_I AND #RETURNED_1_I AND #CYL.SIMULTANEITY_ALARM) OR (NOT (NOT #CYL.ADVANCE_COMMAND AND NOT #ADVANCE) AND #CYL.TIME_EXCEEDED_ALARM AND NOT #ADVANCED_1_I) OR (#ADVANCED_1_ALARM AND NOT "DB2120_MPP_ITC_IPC".RESET_FAULTS)) AND #O_BYTE_0.ADVANCED_INPUT_1 AND "DB1401_PNEUMATIC_SYSTEM".IN_SERVICE;
END_REGION

REGION Network 27: ADVANCED 2 ALARM
   RUNG wire#powerrail
      I_Contact( #CYL.RETURN_COMMAND )
      I_Contact( #"RETURN" )
      Not()
      Contact( #ADVANCED_2_I )
      Contact( #RETURNED_2_I )
      Contact( #CYL.SIMULTANEITY_ALARM )
      wire#w1
      Contact( #O_BYTE_0.ADVANCED_INPUT_2 )
      Contact( "DB1401_PNEUMATIC_SYSTEM".IN_SERVICE )
      Coil( #ADVANCED_2_ALARM )
   END_RUNG
   RUNG wire#powerrail
      I_Contact( #CYL.ADVANCE_COMMAND )
      I_Contact( #ADVANCE )
      Not()
      Contact( #CYL.TIME_EXCEEDED_ALARM )
      I_Contact( #ADVANCED_2_I )
   END_RUNG wire#w1
   RUNG wire#powerrail
      Contact( #ADVANCED_2_ALARM )
      I_Contact( "DB2120_MPP_ITC_IPC".RESET_FAULTS )
   END_RUNG wire#w1
   // the same network as SCL:
   #ADVANCED_2_ALARM := ((NOT (NOT #CYL.RETURN_COMMAND AND NOT #"RETURN") AND #ADVANCED_2_I AND #RETURNED_2_I AND #CYL.SIMULTANEITY_ALARM) OR (NOT (NOT #CYL.ADVANCE_COMMAND AND NOT #ADVANCE) AND #CYL.TIME_EXCEEDED_ALARM AND NOT #ADVANCED_2_I) OR (#ADVANCED_2_ALARM AND NOT "DB2120_MPP_ITC_IPC".RESET_FAULTS)) AND #O_BYTE_0.ADVANCED_INPUT_2 AND "DB1401_PNEUMATIC_SYSTEM".IN_SERVICE;
END_REGION

REGION Network 28: ADVANCED 3 ALARM
   RUNG wire#powerrail
      I_Contact( #CYL.RETURN_COMMAND )
      I_Contact( #"RETURN" )
      Not()
      Contact( #ADVANCED_3_I )
      Contact( #RETURNED_3_I )
      Contact( #CYL.SIMULTANEITY_ALARM )
      wire#w1
      Contact( #O_BYTE_0.ADVANCED_INPUT_3 )
      Contact( "DB1401_PNEUMATIC_SYSTEM".IN_SERVICE )
      Coil( #ADVANCED_3_ALARM )
   END_RUNG
   RUNG wire#powerrail
      I_Contact( #CYL.ADVANCE_COMMAND )
      I_Contact( #ADVANCE )
      Not()
      Contact( #CYL.TIME_EXCEEDED_ALARM )
      I_Contact( #ADVANCED_3_I )
   END_RUNG wire#w1
   RUNG wire#powerrail
      Contact( #ADVANCED_3_ALARM )
      I_Contact( "DB2120_MPP_ITC_IPC".RESET_FAULTS )
   END_RUNG wire#w1
   // the same network as SCL:
   #ADVANCED_3_ALARM := ((NOT (NOT #CYL.RETURN_COMMAND AND NOT #"RETURN") AND #ADVANCED_3_I AND #RETURNED_3_I AND #CYL.SIMULTANEITY_ALARM) OR (NOT (NOT #CYL.ADVANCE_COMMAND AND NOT #ADVANCE) AND #CYL.TIME_EXCEEDED_ALARM AND NOT #ADVANCED_3_I) OR (#ADVANCED_3_ALARM AND NOT "DB2120_MPP_ITC_IPC".RESET_FAULTS)) AND #O_BYTE_0.ADVANCED_INPUT_3 AND "DB1401_PNEUMATIC_SYSTEM".IN_SERVICE;
END_REGION

REGION Network 29: ADVANCED 4 ALARM
   RUNG wire#powerrail
      I_Contact( #CYL.RETURN_COMMAND )
      I_Contact( #"RETURN" )
      Not()
      Contact( #ADVANCED_4_I )
      Contact( #RETURNED_4_I )
      Contact( #CYL.SIMULTANEITY_ALARM )
      wire#w1
      Contact( #O_BYTE_0.ADVANCED_INPUT_4 )
      Contact( "DB1401_PNEUMATIC_SYSTEM".IN_SERVICE )
      Coil( #ADVANCED_4_ALARM )
   END_RUNG
   RUNG wire#powerrail
      I_Contact( #CYL.ADVANCE_COMMAND )
      I_Contact( #ADVANCE )
      Not()
      Contact( #CYL.TIME_EXCEEDED_ALARM )
      I_Contact( #ADVANCED_4_I )
   END_RUNG wire#w1
   RUNG wire#powerrail
      Contact( #ADVANCED_4_ALARM )
      I_Contact( "DB2120_MPP_ITC_IPC".RESET_FAULTS )
   END_RUNG wire#w1
   // the same network as SCL:
   #ADVANCED_4_ALARM := ((NOT (NOT #CYL.RETURN_COMMAND AND NOT #"RETURN") AND #ADVANCED_4_I AND #RETURNED_4_I AND #CYL.SIMULTANEITY_ALARM) OR (NOT (NOT #CYL.ADVANCE_COMMAND AND NOT #ADVANCE) AND #CYL.TIME_EXCEEDED_ALARM AND NOT #ADVANCED_4_I) OR (#ADVANCED_4_ALARM AND NOT "DB2120_MPP_ITC_IPC".RESET_FAULTS)) AND #O_BYTE_0.ADVANCED_INPUT_4 AND "DB1401_PNEUMATIC_SYSTEM".IN_SERVICE;
END_REGION

REGION Network 30: RETURNED 1 ALARM
   RUNG wire#powerrail
      I_Contact( #CYL.ADVANCE_COMMAND )
      I_Contact( #ADVANCE )
      Not()
      Contact( #ADVANCED_1_I )
      Contact( #RETURNED_1_I )
      Contact( #CYL.SIMULTANEITY_ALARM )
      wire#w1
      Contact( #O_BYTE_0.RETURNED_INPUT_1 )
      Contact( "DB1401_PNEUMATIC_SYSTEM".IN_SERVICE )
      Coil( #RETURNED_1_ALARM )
   END_RUNG
   RUNG wire#powerrail
      I_Contact( #CYL.RETURN_COMMAND )
      I_Contact( #"RETURN" )
      Not()
      Contact( #CYL.TIME_EXCEEDED_ALARM )
      I_Contact( #RETURNED_1_I )
   END_RUNG wire#w1
   RUNG wire#powerrail
      Contact( #RETURNED_1_ALARM )
      I_Contact( "DB2120_MPP_ITC_IPC".RESET_FAULTS )
   END_RUNG wire#w1
   // the same network as SCL:
   #RETURNED_1_ALARM := ((NOT (NOT #CYL.ADVANCE_COMMAND AND NOT #ADVANCE) AND #ADVANCED_1_I AND #RETURNED_1_I AND #CYL.SIMULTANEITY_ALARM) OR (NOT (NOT #CYL.RETURN_COMMAND AND NOT #"RETURN") AND #CYL.TIME_EXCEEDED_ALARM AND NOT #RETURNED_1_I) OR (#RETURNED_1_ALARM AND NOT "DB2120_MPP_ITC_IPC".RESET_FAULTS)) AND #O_BYTE_0.RETURNED_INPUT_1 AND "DB1401_PNEUMATIC_SYSTEM".IN_SERVICE;
END_REGION

REGION Network 31: RETURNED 2 ALARM
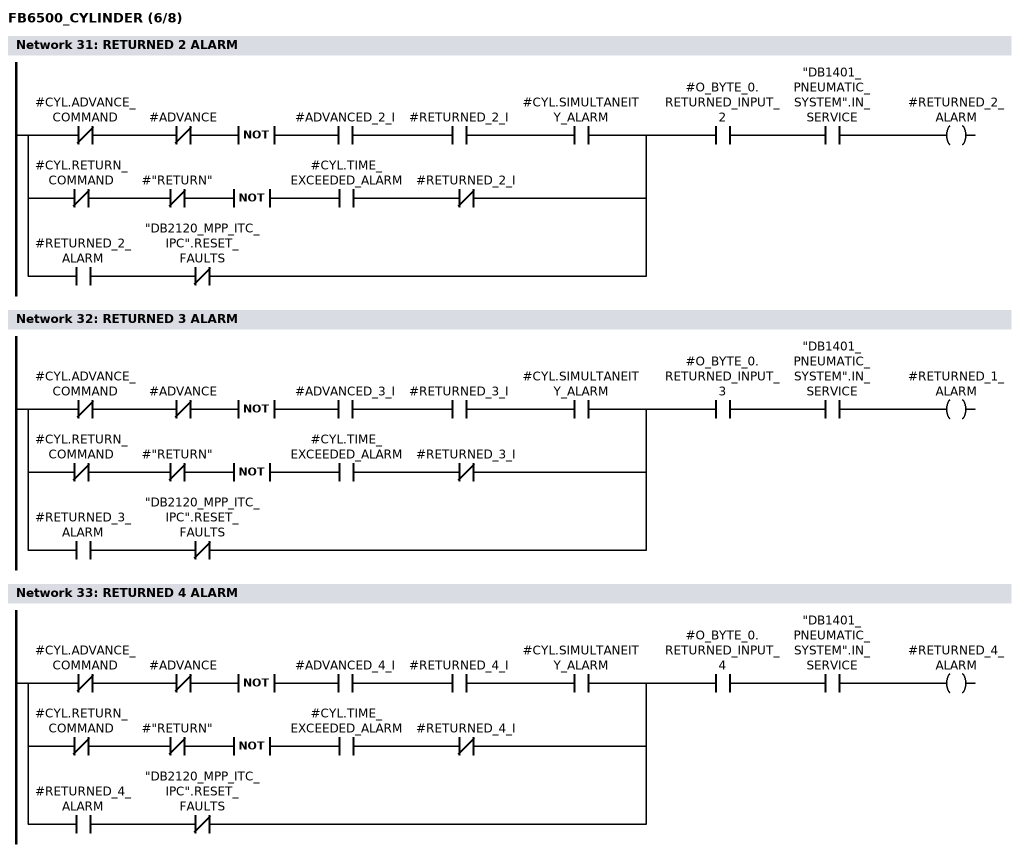
   RUNG wire#powerrail
      I_Contact( #CYL.ADVANCE_COMMAND )
      I_Contact( #ADVANCE )
      Not()
      Contact( #ADVANCED_2_I )
      Contact( #RETURNED_2_I )
      Contact( #CYL.SIMULTANEITY_ALARM )
      wire#w1
      Contact( #O_BYTE_0.RETURNED_INPUT_2 )
      Contact( "DB1401_PNEUMATIC_SYSTEM".IN_SERVICE )
      Coil( #RETURNED_2_ALARM )
   END_RUNG
   RUNG wire#powerrail
      I_Contact( #CYL.RETURN_COMMAND )
      I_Contact( #"RETURN" )
      Not()
      Contact( #CYL.TIME_EXCEEDED_ALARM )
      I_Contact( #RETURNED_2_I )
   END_RUNG wire#w1
   RUNG wire#powerrail
      Contact( #RETURNED_2_ALARM )
      I_Contact( "DB2120_MPP_ITC_IPC".RESET_FAULTS )
   END_RUNG wire#w1
   // the same network as SCL:
   #RETURNED_2_ALARM := ((NOT (NOT #CYL.ADVANCE_COMMAND AND NOT #ADVANCE) AND #ADVANCED_2_I AND #RETURNED_2_I AND #CYL.SIMULTANEITY_ALARM) OR (NOT (NOT #CYL.RETURN_COMMAND AND NOT #"RETURN") AND #CYL.TIME_EXCEEDED_ALARM AND NOT #RETURNED_2_I) OR (#RETURNED_2_ALARM AND NOT "DB2120_MPP_ITC_IPC".RESET_FAULTS)) AND #O_BYTE_0.RETURNED_INPUT_2 AND "DB1401_PNEUMATIC_SYSTEM".IN_SERVICE;
END_REGION

REGION Network 32: RETURNED 3 ALARM
   RUNG wire#powerrail
      I_Contact( #CYL.ADVANCE_COMMAND )
      I_Contact( #ADVANCE )
      Not()
      Contact( #ADVANCED_3_I )
      Contact( #RETURNED_3_I )
      Contact( #CYL.SIMULTANEITY_ALARM )
      wire#w1
      Contact( #O_BYTE_0.RETURNED_INPUT_3 )
      Contact( "DB1401_PNEUMATIC_SYSTEM".IN_SERVICE )
      Coil( #RETURNED_1_ALARM )
   END_RUNG
   RUNG wire#powerrail
      I_Contact( #CYL.RETURN_COMMAND )
      I_Contact( #"RETURN" )
      Not()
      Contact( #CYL.TIME_EXCEEDED_ALARM )
      I_Contact( #RETURNED_3_I )
   END_RUNG wire#w1
   RUNG wire#powerrail
      Contact( #RETURNED_3_ALARM )
      I_Contact( "DB2120_MPP_ITC_IPC".RESET_FAULTS )
   END_RUNG wire#w1
   // the same network as SCL:
   #RETURNED_1_ALARM := ((NOT (NOT #CYL.ADVANCE_COMMAND AND NOT #ADVANCE) AND #ADVANCED_3_I AND #RETURNED_3_I AND #CYL.SIMULTANEITY_ALARM) OR (NOT (NOT #CYL.RETURN_COMMAND AND NOT #"RETURN") AND #CYL.TIME_EXCEEDED_ALARM AND NOT #RETURNED_3_I) OR (#RETURNED_3_ALARM AND NOT "DB2120_MPP_ITC_IPC".RESET_FAULTS)) AND #O_BYTE_0.RETURNED_INPUT_3 AND "DB1401_PNEUMATIC_SYSTEM".IN_SERVICE;
END_REGION

REGION Network 33: RETURNED 4 ALARM
   RUNG wire#powerrail
      I_Contact( #CYL.ADVANCE_COMMAND )
      I_Contact( #ADVANCE )
      Not()
      Contact( #ADVANCED_4_I )
      Contact( #RETURNED_4_I )
      Contact( #CYL.SIMULTANEITY_ALARM )
      wire#w1
      Contact( #O_BYTE_0.RETURNED_INPUT_4 )
      Contact( "DB1401_PNEUMATIC_SYSTEM".IN_SERVICE )
      Coil( #RETURNED_4_ALARM )
   END_RUNG
   RUNG wire#powerrail
      I_Contact( #CYL.RETURN_COMMAND )
      I_Contact( #"RETURN" )
      Not()
      Contact( #CYL.TIME_EXCEEDED_ALARM )
      I_Contact( #RETURNED_4_I )
   END_RUNG wire#w1
   RUNG wire#powerrail
      Contact( #RETURNED_4_ALARM )
      I_Contact( "DB2120_MPP_ITC_IPC".RESET_FAULTS )
   END_RUNG wire#w1
   // the same network as SCL:
   #RETURNED_4_ALARM := ((NOT (NOT #CYL.ADVANCE_COMMAND AND NOT #ADVANCE) AND #ADVANCED_4_I AND #RETURNED_4_I AND #CYL.SIMULTANEITY_ALARM) OR (NOT (NOT #CYL.RETURN_COMMAND AND NOT #"RETURN") AND #CYL.TIME_EXCEEDED_ALARM AND NOT #RETURNED_4_I) OR (#RETURNED_4_ALARM AND NOT "DB2120_MPP_ITC_IPC".RESET_FAULTS)) AND #O_BYTE_0.RETURNED_INPUT_4 AND "DB1401_PNEUMATIC_SYSTEM".IN_SERVICE;
END_REGION

REGION Network 34: IMMEDIATE STOP AND STOP END OF CYCLE ALARMS
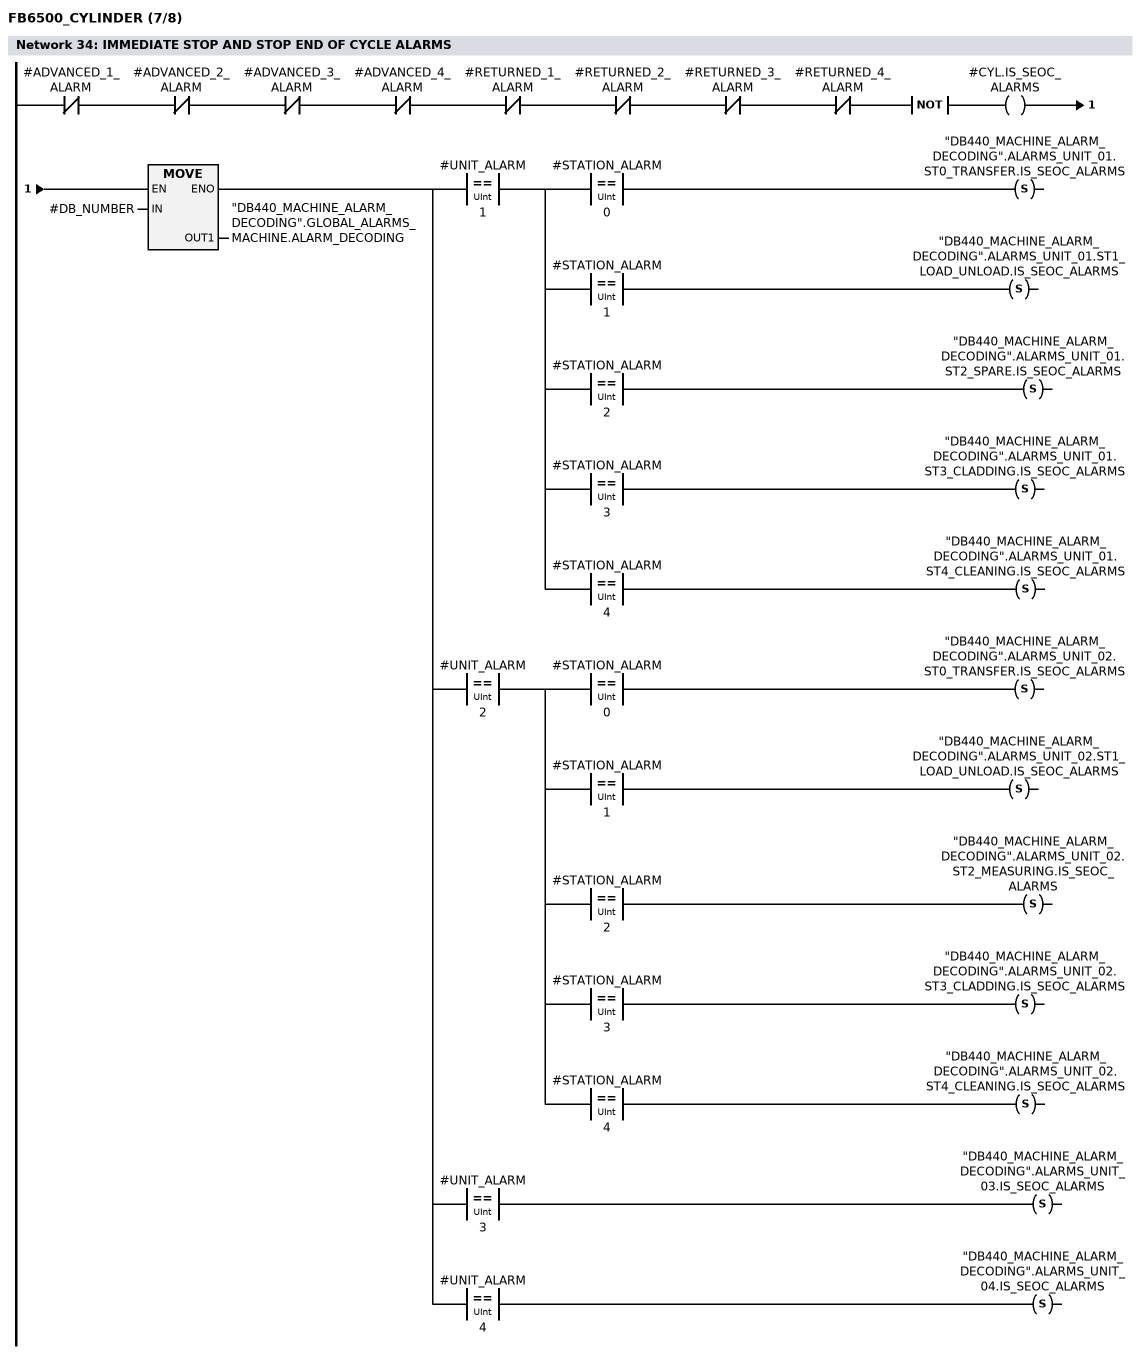
   RUNG wire#powerrail
      I_Contact( #ADVANCED_1_ALARM )
      I_Contact( #ADVANCED_2_ALARM )
      I_Contact( #ADVANCED_3_ALARM )
      I_Contact( #ADVANCED_4_ALARM )
      I_Contact( #RETURNED_1_ALARM )
      I_Contact( #RETURNED_2_ALARM )
      I_Contact( #RETURNED_3_ALARM )
      I_Contact( #RETURNED_4_ALARM )
      Not()
      Coil( #CYL.IS_SEOC_ALARMS )
      { S7_GenerateENO := "TRUE" } Move(in := #DB_NUMBER, out1 => "DB440_MACHINE_ALARM_DECODING".GLOBAL_ALARMS_MACHINE.ALARM_DECODING)
      wire#w1
      { S7_Templates := "SrcType := UInt" } EQ_Contact(in1 := #UNIT_ALARM, in2 := 1)
      wire#w2
      { S7_Templates := "SrcType := UInt" } EQ_Contact(in1 := #STATION_ALARM, in2 := 0)
      S_Coil( "DB440_MACHINE_ALARM_DECODING".ALARMS_UNIT_01.ST0_TRANSFER.IS_SEOC_ALARMS )
   END_RUNG
   RUNG wire#w2
      { S7_Templates := "SrcType := UInt" } EQ_Contact(in1 := #STATION_ALARM, in2 := 1)
      S_Coil( "DB440_MACHINE_ALARM_DECODING".ALARMS_UNIT_01.ST1_LOAD_UNLOAD.IS_SEOC_ALARMS )
   END_RUNG
   RUNG wire#w2
      { S7_Templates := "SrcType := UInt" } EQ_Contact(in1 := #STATION_ALARM, in2 := 2)
      S_Coil( "DB440_MACHINE_ALARM_DECODING".ALARMS_UNIT_01.ST2_SPARE.IS_SEOC_ALARMS )
   END_RUNG
   RUNG wire#w2
      { S7_Templates := "SrcType := UInt" } EQ_Contact(in1 := #STATION_ALARM, in2 := 3)
      S_Coil( "DB440_MACHINE_ALARM_DECODING".ALARMS_UNIT_01.ST3_CLADDING.IS_SEOC_ALARMS )
   END_RUNG
   RUNG wire#w2
      { S7_Templates := "SrcType := UInt" } EQ_Contact(in1 := #STATION_ALARM, in2 := 4)
      S_Coil( "DB440_MACHINE_ALARM_DECODING".ALARMS_UNIT_01.ST4_CLEANING.IS_SEOC_ALARMS )
   END_RUNG
   RUNG wire#w1
      { S7_Templates := "SrcType := UInt" } EQ_Contact(in1 := #UNIT_ALARM, in2 := 2)
      wire#w3
      { S7_Templates := "SrcType := UInt" } EQ_Contact(in1 := #STATION_ALARM, in2 := 0)
      S_Coil( "DB440_MACHINE_ALARM_DECODING".ALARMS_UNIT_02.ST0_TRANSFER.IS_SEOC_ALARMS )
   END_RUNG
   RUNG wire#w3
      { S7_Templates := "SrcType := UInt" } EQ_Contact(in1 := #STATION_ALARM, in2 := 1)
      S_Coil( "DB440_MACHINE_ALARM_DECODING".ALARMS_UNIT_02.ST1_LOAD_UNLOAD.IS_SEOC_ALARMS )
   END_RUNG
   RUNG wire#w3
      { S7_Templates := "SrcType := UInt" } EQ_Contact(in1 := #STATION_ALARM, in2 := 2)
      S_Coil( "DB440_MACHINE_ALARM_DECODING".ALARMS_UNIT_02.ST2_MEASURING.IS_SEOC_ALARMS )
   END_RUNG
   RUNG wire#w3
      { S7_Templates := "SrcType := UInt" } EQ_Contact(in1 := #STATION_ALARM, in2 := 3)
      S_Coil( "DB440_MACHINE_ALARM_DECODING".ALARMS_UNIT_02.ST3_CLADDING.IS_SEOC_ALARMS )
   END_RUNG
   RUNG wire#w3
      { S7_Templates := "SrcType := UInt" } EQ_Contact(in1 := #STATION_ALARM, in2 := 4)
      S_Coil( "DB440_MACHINE_ALARM_DECODING".ALARMS_UNIT_02.ST4_CLEANING.IS_SEOC_ALARMS )
   END_RUNG
   RUNG wire#w1
      { S7_Templates := "SrcType := UInt" } EQ_Contact(in1 := #UNIT_ALARM, in2 := 3)
      S_Coil( "DB440_MACHINE_ALARM_DECODING".ALARMS_UNIT_03.IS_SEOC_ALARMS )
   END_RUNG
   RUNG wire#w1
      { S7_Templates := "SrcType := UInt" } EQ_Contact(in1 := #UNIT_ALARM, in2 := 4)
      S_Coil( "DB440_MACHINE_ALARM_DECODING".ALARMS_UNIT_04.IS_SEOC_ALARMS )
   END_RUNG
   // the same network as SCL:
   // ENO of a box is taken as its EN; it also drops when the box reports an error
   #CYL.IS_SEOC_ALARMS := NOT (NOT #ADVANCED_1_ALARM AND NOT #ADVANCED_2_ALARM AND NOT #ADVANCED_3_ALARM AND NOT #ADVANCED_4_ALARM AND NOT #RETURNED_1_ALARM AND NOT #RETURNED_2_ALARM AND NOT #RETURNED_3_ALARM AND NOT #RETURNED_4_ALARM);
   IF #CYL.IS_SEOC_ALARMS THEN
       "DB440_MACHINE_ALARM_DECODING".GLOBAL_ALARMS_MACHINE.ALARM_DECODING := #DB_NUMBER;
   END_IF;
   #_w1 := #CYL.IS_SEOC_ALARMS AND (#UNIT_ALARM = 1);
   IF #_w1 AND (#STATION_ALARM = 0) THEN
       "DB440_MACHINE_ALARM_DECODING".ALARMS_UNIT_01.ST0_TRANSFER.IS_SEOC_ALARMS := TRUE;
   END_IF;
   IF #_w1 AND (#STATION_ALARM = 1) THEN
       "DB440_MACHINE_ALARM_DECODING".ALARMS_UNIT_01.ST1_LOAD_UNLOAD.IS_SEOC_ALARMS := TRUE;
   END_IF;
   IF #_w1 AND (#STATION_ALARM = 2) THEN
       "DB440_MACHINE_ALARM_DECODING".ALARMS_UNIT_01.ST2_SPARE.IS_SEOC_ALARMS := TRUE;
   END_IF;
   IF #_w1 AND (#STATION_ALARM = 3) THEN
       "DB440_MACHINE_ALARM_DECODING".ALARMS_UNIT_01.ST3_CLADDING.IS_SEOC_ALARMS := TRUE;
   END_IF;
   IF #_w1 AND (#STATION_ALARM = 4) THEN
       "DB440_MACHINE_ALARM_DECODING".ALARMS_UNIT_01.ST4_CLEANING.IS_SEOC_ALARMS := TRUE;
   END_IF;
   #_w2 := #CYL.IS_SEOC_ALARMS AND (#UNIT_ALARM = 2);
   IF #_w2 AND (#STATION_ALARM = 0) THEN
       "DB440_MACHINE_ALARM_DECODING".ALARMS_UNIT_02.ST0_TRANSFER.IS_SEOC_ALARMS := TRUE;
   END_IF;
   IF #_w2 AND (#STATION_ALARM = 1) THEN
       "DB440_MACHINE_ALARM_DECODING".ALARMS_UNIT_02.ST1_LOAD_UNLOAD.IS_SEOC_ALARMS := TRUE;
   END_IF;
   IF #_w2 AND (#STATION_ALARM = 2) THEN
       "DB440_MACHINE_ALARM_DECODING".ALARMS_UNIT_02.ST2_MEASURING.IS_SEOC_ALARMS := TRUE;
   END_IF;
   IF #_w2 AND (#STATION_ALARM = 3) THEN
       "DB440_MACHINE_ALARM_DECODING".ALARMS_UNIT_02.ST3_CLADDING.IS_SEOC_ALARMS := TRUE;
   END_IF;
   IF #_w2 AND (#STATION_ALARM = 4) THEN
       "DB440_MACHINE_ALARM_DECODING".ALARMS_UNIT_02.ST4_CLEANING.IS_SEOC_ALARMS := TRUE;
   END_IF;
   IF #CYL.IS_SEOC_ALARMS AND (#UNIT_ALARM = 3) THEN
       "DB440_MACHINE_ALARM_DECODING".ALARMS_UNIT_03.IS_SEOC_ALARMS := TRUE;
   END_IF;
   IF #CYL.IS_SEOC_ALARMS AND (#UNIT_ALARM = 4) THEN
       "DB440_MACHINE_ALARM_DECODING".ALARMS_UNIT_04.IS_SEOC_ALARMS := TRUE;
   END_IF;
END_REGION

REGION Network 35: ANY ACTIVE ALARM
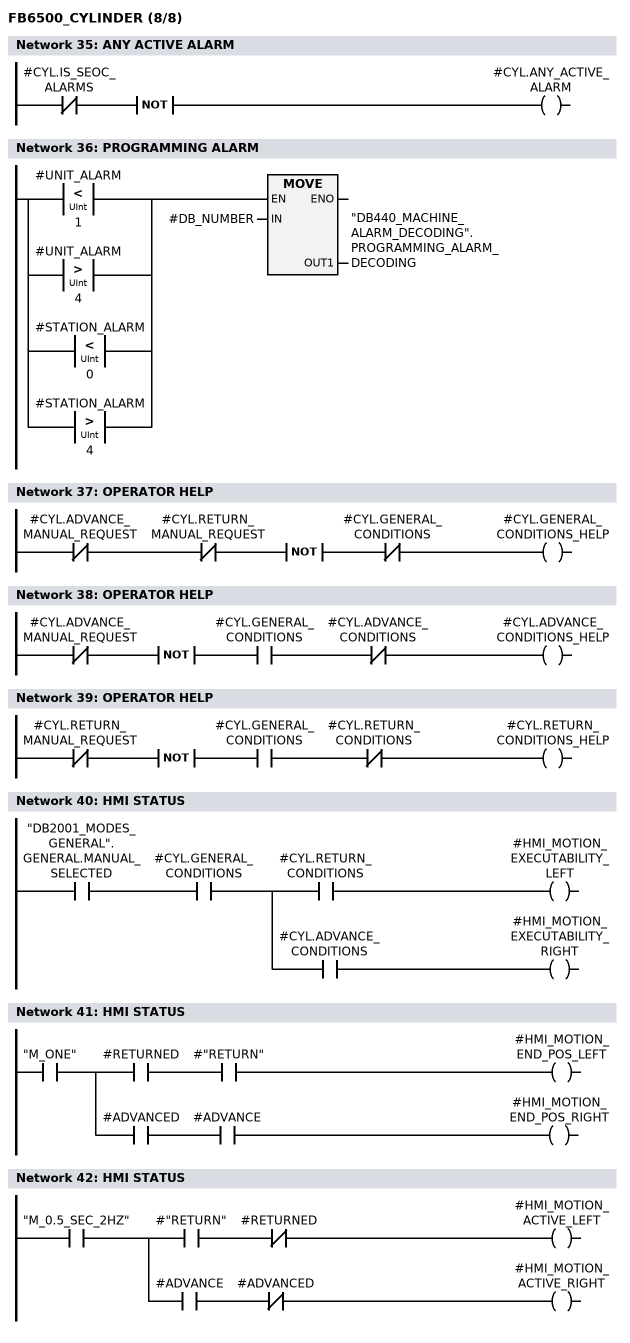
   RUNG wire#powerrail
      I_Contact( #CYL.IS_SEOC_ALARMS )
      Not()
      Coil( #CYL.ANY_ACTIVE_ALARM )
   END_RUNG
   // the same network as SCL:
   #CYL.ANY_ACTIVE_ALARM := NOT (NOT #CYL.IS_SEOC_ALARMS);
END_REGION

REGION Network 36: PROGRAMMING ALARM
   RUNG wire#powerrail
      { S7_Templates := "SrcType := UInt" } LT_Contact(in1 := #UNIT_ALARM, in2 := 1)
      wire#w1
      Move(in := #DB_NUMBER, out1 => "DB440_MACHINE_ALARM_DECODING".PROGRAMMING_ALARM_DECODING)
   END_RUNG
   RUNG wire#powerrail
      { S7_Templates := "SrcType := UInt" } GT_Contact(in1 := #UNIT_ALARM, in2 := 4)
   END_RUNG wire#w1
   RUNG wire#powerrail
      { S7_Templates := "SrcType := UInt" } LT_Contact(in1 := #STATION_ALARM, in2 := 0)
   END_RUNG wire#w1
   RUNG wire#powerrail
      { S7_Templates := "SrcType := UInt" } GT_Contact(in1 := #STATION_ALARM, in2 := 4)
   END_RUNG wire#w1
   // the same network as SCL:
   IF (#UNIT_ALARM < 1) OR (#UNIT_ALARM > 4) OR (#STATION_ALARM < 0) OR (#STATION_ALARM > 4) THEN
       "DB440_MACHINE_ALARM_DECODING".PROGRAMMING_ALARM_DECODING := #DB_NUMBER;
   END_IF;
END_REGION

REGION Network 37: OPERATOR HELP
   RUNG wire#powerrail
      I_Contact( #CYL.ADVANCE_MANUAL_REQUEST )
      I_Contact( #CYL.RETURN_MANUAL_REQUEST )
      Not()
      I_Contact( #CYL.GENERAL_CONDITIONS )
      Coil( #CYL.GENERAL_CONDITIONS_HELP )
   END_RUNG
   // the same network as SCL:
   #CYL.GENERAL_CONDITIONS_HELP := NOT (NOT #CYL.ADVANCE_MANUAL_REQUEST AND NOT #CYL.RETURN_MANUAL_REQUEST) AND NOT #CYL.GENERAL_CONDITIONS;
END_REGION

REGION Network 38: OPERATOR HELP
   RUNG wire#powerrail
      I_Contact( #CYL.ADVANCE_MANUAL_REQUEST )
      Not()
      Contact( #CYL.GENERAL_CONDITIONS )
      I_Contact( #CYL.ADVANCE_CONDITIONS )
      Coil( #CYL.ADVANCE_CONDITIONS_HELP )
   END_RUNG
   // the same network as SCL:
   #CYL.ADVANCE_CONDITIONS_HELP := NOT (NOT #CYL.ADVANCE_MANUAL_REQUEST) AND #CYL.GENERAL_CONDITIONS AND NOT #CYL.ADVANCE_CONDITIONS;
END_REGION

REGION Network 39: OPERATOR HELP
   RUNG wire#powerrail
      I_Contact( #CYL.RETURN_MANUAL_REQUEST )
      Not()
      Contact( #CYL.GENERAL_CONDITIONS )
      I_Contact( #CYL.RETURN_CONDITIONS )
      Coil( #CYL.RETURN_CONDITIONS_HELP )
   END_RUNG
   // the same network as SCL:
   #CYL.RETURN_CONDITIONS_HELP := NOT (NOT #CYL.RETURN_MANUAL_REQUEST) AND #CYL.GENERAL_CONDITIONS AND NOT #CYL.RETURN_CONDITIONS;
END_REGION

REGION Network 40: HMI STATUS
   RUNG wire#powerrail
      Contact( "DB2001_MODES_GENERAL".GENERAL.MANUAL_SELECTED )
      Contact( #CYL.GENERAL_CONDITIONS )
      wire#w1
      Contact( #CYL.RETURN_CONDITIONS )
      Coil( #HMI_MOTION_EXECUTABILITY_LEFT )
   END_RUNG
   RUNG wire#w1
      Contact( #CYL.ADVANCE_CONDITIONS )
      Coil( #HMI_MOTION_EXECUTABILITY_RIGHT )
   END_RUNG
   // the same network as SCL:
   #_w1 := "DB2001_MODES_GENERAL".GENERAL.MANUAL_SELECTED AND #CYL.GENERAL_CONDITIONS;
   #HMI_MOTION_EXECUTABILITY_LEFT := #_w1 AND #CYL.RETURN_CONDITIONS;
   #HMI_MOTION_EXECUTABILITY_RIGHT := #_w1 AND #CYL.ADVANCE_CONDITIONS;
END_REGION

REGION Network 41: HMI STATUS
   RUNG wire#powerrail
      Contact( "M_ONE" )
      wire#w1
      Contact( #RETURNED )
      Contact( #"RETURN" )
      Coil( #HMI_MOTION_END_POS_LEFT )
   END_RUNG
   RUNG wire#w1
      Contact( #ADVANCED )
      Contact( #ADVANCE )
      Coil( #HMI_MOTION_END_POS_RIGHT )
   END_RUNG
   // the same network as SCL:
   #HMI_MOTION_END_POS_LEFT := "M_ONE" AND #RETURNED AND #"RETURN";
   #HMI_MOTION_END_POS_RIGHT := "M_ONE" AND #ADVANCED AND #ADVANCE;
END_REGION

REGION Network 42: HMI STATUS
   RUNG wire#powerrail
      Contact( "M_0.5_SEC_2HZ" )
      wire#w1
      Contact( #"RETURN" )
      I_Contact( #RETURNED )
      Coil( #HMI_MOTION_ACTIVE_LEFT )
   END_RUNG
   RUNG wire#w1
      Contact( #ADVANCE )
      I_Contact( #ADVANCED )
      Coil( #HMI_MOTION_ACTIVE_RIGHT )
   END_RUNG
   // the same network as SCL:
   #HMI_MOTION_ACTIVE_LEFT := "M_0.5_SEC_2HZ" AND #"RETURN" AND NOT #RETURNED;
   #HMI_MOTION_ACTIVE_RIGHT := "M_0.5_SEC_2HZ" AND #ADVANCE AND NOT #ADVANCED;
END_REGION
END_FUNCTION_BLOCK
